FUNCTION F_LIN : REAL
VAR_INPUT
	X : REAL;
	A : REAL;
	B : REAL;
END_VAR


(*
version 1.0	1 sep 2006
programmer 	hugo
tested by		tobias

this function calculates the linear equation f_lin = a*x + b

*)


F_lin := A * X + B;

END_FUNCTION

(* stored: Version 1.1.0.1
   POU F_LIN: Id {952a72b5-e8a1-4914-988b-b5c29b4c32cb}, SpecialFunc None *)
